FUNCTION_BLOCK Forces2
VAR_INPUT
END_VAR
VAR_OUTPUT
END_VAR
VAR
END_VAR

END_FUNCTION_BLOCK

(* stored: Version 1.1.0.1, ProductVersion 3.1.4024.11
   POU Forces2: Id {ab65772c-f89c-4b17-a551-a19d9cbf8774}, SpecialFunc None *)
